ABB RobotStudio station: Modulo_2.rspag

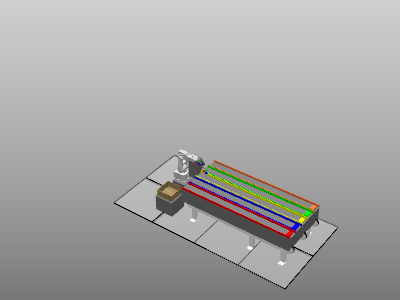
--- station ---
Station Project2 (saved by RobotStudio 25.1.11133.0)
Controller Controlador1, task T_ROB1: task frame (RAPID world) sits at (0, 0, 437.58) mm in the station
Controller Controlador1
  mechanical unit ROB_1: IRB120_3_58__01, 6 joints, base frame (0, 0, 0) mm
Layout (positions relative to the parent item):
  - IRB120_3_58__01 [mechanism, from %ABB.RobotStudio.Models.IRB120%\IRB120_3_58_G_01.rslib] at (0, 0, 437.58) mm; joint values [0, 0, 0, 0, 0.5236, 0] (rad or m)
  - MyTool [mechanism, from Training Objects\myTool.rslib] at (364.35, 0, 1031.58) mm, rotated rx 180 ry 60 rz 180 deg
  - Conveyor [part, from %ABB.RobotStudio.Models.Conveyors%\Conveyor 2400 3str h2.rslib] at (479.82, -405.8, 0) mm
  - Base Robot [graphiccomponentgroup]
    - Pieza_1 [part] at (-150, -150, 0) mm, size 300 x 300 x 200 mm
    - Pieza_2 [part], size 300 x 300 x 237.6 mm
  - Caja [part] at (0, 0, 145) mm, size 350 x 350 x 150 mm
  - Estropajo_Morado [part] at (2649.97, 391.91, 691.61) mm, size 80 x 120 x 43 mm
  - Estropajo_Verde [part] at (2649.97, 171.91, 691.61) mm, size 80 x 120 x 43 mm
  - Estropajo_Amarillo [part, from Components\Estropajo_6.rslib] at (2649.97, -48.09, 691.61) mm
  - Estropajo_Azul [part] at (2649.97, -268.09, 691.61) mm, size 80 x 120 x 43 mm
  - Estropajo_Rojo [part] at (2649.97, -488.09, 691.61) mm, size 80 x 120 x 43 mm
  - Base Caja [graphiccomponentgroup]
    - Base Caja [part] at (-190.34, -650.22, 0) mm, size 400 x 400 x 350 mm
  - LinearMover2 [smart component, from Components\LinearMover2.rslib]
      properties: Object=(none); Direction=[-0.001 0 0]; Distance=2.2; Duration=2; Reference=Global; ReferenceObject=(none)
  - LinearMover2_2 [smart component, from Components\LinearMover2.rslib]
      properties: Object=(none); Direction=[-0.001 0 0]; Distance=2.2; Duration=2; Reference=Global; ReferenceObject=(none)
  - LinearMover2_3 [smart component, from Components\LinearMover2.rslib]
      properties: Object=(none); Direction=[-0.001 0 0]; Distance=2.2; Duration=2; Reference=Global; ReferenceObject=(none)
  - LinearMover2_4 [smart component, from Components\LinearMover2.rslib]
      properties: Object=(none); Direction=[-0.001 0 0]; Distance=2.2; Duration=2; Reference=Global; ReferenceObject=(none)
  - LinearMover2_5 [smart component, from Components\LinearMover2.rslib]
      properties: Object=(none); Direction=[-0.001 0 0]; Distance=2.2; Duration=2; Reference=Global; ReferenceObject=(none)
  - Source [smart component, from Components\Source.rslib]
      properties: Source=Estropajo_Rojo; Copy=(none); Parent=(none); Position=[2.649968 -0.488094 0.691615]; Orientation=[0 0 0]; Transient=true; PhysicsBehavior=-1
  - Source_2 [smart component, from Components\Source.rslib]
      properties: Source=Estropajo_Azul; Copy=(none); Parent=(none); Position=[2.649968 -0.268094 0.691615]; Orientation=[0 0 0]; Transient=true; PhysicsBehavior=-1
  - Source_3 [smart component, from Components\Source.rslib]
      properties: Source=Estropajo_Amarillo; Copy=(none); Parent=(none); Position=[2.649968 -0.048094 0.691615]; Orientation=[0 0 0]; Transient=true; PhysicsBehavior=-1
  - Source_4 [smart component, from Components\Source.rslib]
      properties: Source=Estropajo_Verde; Copy=(none); Parent=(none); Position=[2.649968 0.171906 0.691615]; Orientation=[0 0 0]; Transient=true; PhysicsBehavior=-1
  - Source_5 [smart component, from Components\Source.rslib]
      properties: Source=Estropajo_Morado; Copy=(none); Parent=(none); Position=[2.649968 0.391906 0.691615]; Orientation=[0 0 0]; Transient=true; PhysicsBehavior=-1
  - Base Apilar [part], size 200 x 200 x 700 mm
  - Attacher [smart component, from Components\Attacher.rslib]
      properties: Parent=MyTool; Flange=0; Child=(none); Mount=false; Offset=[0 0 0]; Orientation=[0 0 0]
  - Attacher_2 [smart component, from Components\Attacher.rslib]
      properties: Parent=MyTool; Flange=0; Child=(none); Mount=false; Offset=[0 0 0]; Orientation=[0 0 0]
  - Attacher_3 [smart component, from Components\Attacher.rslib]
      properties: Parent=MyTool; Flange=0; Child=(none); Mount=false; Offset=[0 0 0]; Orientation=[0 0 0]
  - Attacher_4 [smart component, from Components\Attacher.rslib]
      properties: Parent=MyTool; Flange=0; Child=(none); Mount=false; Offset=[0 0 0]; Orientation=[0 0 0]
  - Attacher_5 [smart component, from Components\Attacher.rslib]
      properties: Parent=MyTool; Flange=0; Child=(none); Mount=false; Offset=[0 0 0]; Orientation=[0 0 0]
  - Detacher [smart component, from Components\Detacher.rslib]
      properties: Child=(none); KeepPosition=true
  - Detacher_2 [smart component, from Components\Detacher.rslib]
      properties: Child=(none); KeepPosition=true
  - Detacher_3 [smart component, from Components\Detacher.rslib]
      properties: Child=(none); KeepPosition=true
  - Detacher_4 [smart component, from Components\Detacher.rslib]
      properties: Child=(none); KeepPosition=true
  - Detacher_5 [smart component, from Components\Detacher.rslib]
      properties: Child=(none); KeepPosition=true
  - Cinta salida_2 [part, from Components\Cinta salida.rslib] at (2961.89, -775, 0) mm
Attachment: MyTool is attached to IRB120_3_58__01 / Link6
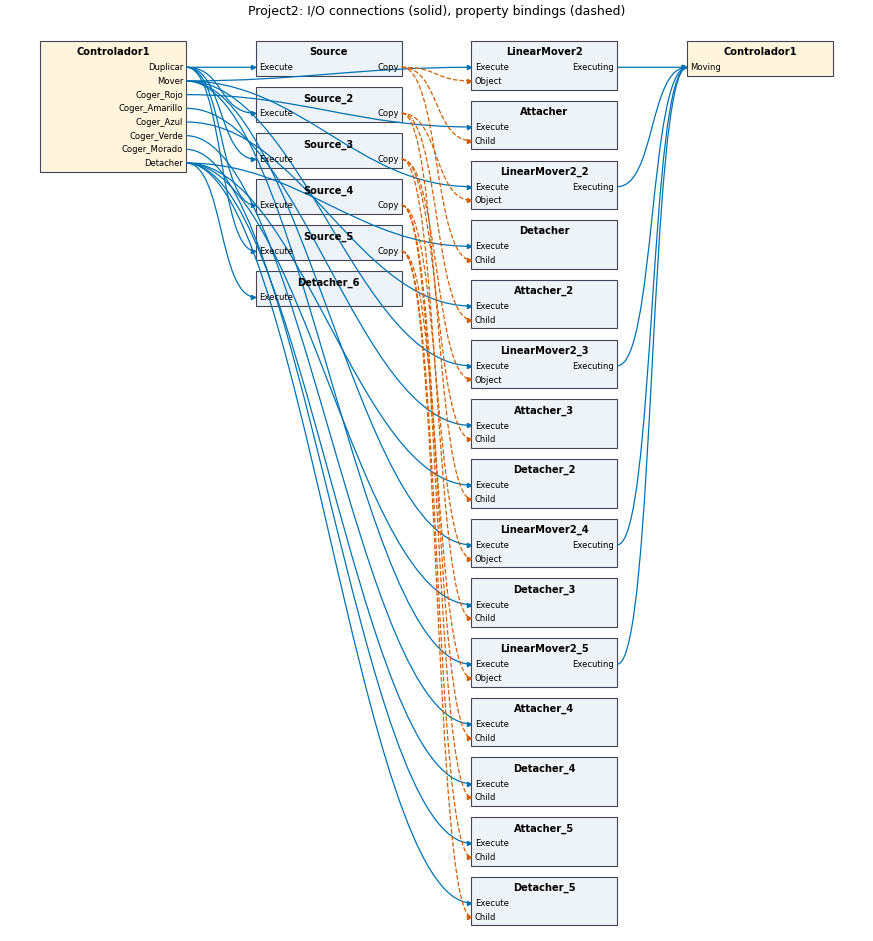
Station logic (signal -> signal, property => property):
  Controlador1.Duplicar -> Source.Execute
  Controlador1.Duplicar -> Source_2.Execute
  Controlador1.Duplicar -> Source_3.Execute
  Controlador1.Duplicar -> Source_4.Execute
  Controlador1.Duplicar -> Source_5.Execute
  Controlador1.Mover -> LinearMover2.Execute
  Controlador1.Mover -> LinearMover2_2.Execute
  Controlador1.Mover -> LinearMover2_3.Execute
  Controlador1.Mover -> LinearMover2_4.Execute
  Controlador1.Mover -> LinearMover2_5.Execute
  Controlador1.Coger_Rojo -> Attacher.Execute
  Controlador1.Coger_Amarillo -> Attacher_3.Execute
  Controlador1.Coger_Azul -> Attacher_2.Execute
  Controlador1.Coger_Verde -> Attacher_4.Execute
  Controlador1.Coger_Morado -> Attacher_5.Execute
  Controlador1.Detacher -> Detacher.Execute
  Controlador1.Detacher -> Detacher_2.Execute
  Controlador1.Detacher -> Detacher_3.Execute
  Controlador1.Detacher -> Detacher_4.Execute
  Controlador1.Detacher -> Detacher_5.Execute
  LinearMover2.Executing -> Controlador1.Moving
  LinearMover2_3.Executing -> Controlador1.Moving
  LinearMover2_5.Executing -> Controlador1.Moving
  LinearMover2_2.Executing -> Controlador1.Moving
  LinearMover2_4.Executing -> Controlador1.Moving
  Controlador1.Detacher -> Detacher_6.Execute
  Source.Copy => LinearMover2.Object
  Source_5.Copy => LinearMover2_5.Object
  Source_2.Copy => LinearMover2_2.Object
  Source_3.Copy => LinearMover2_3.Object
  Source_4.Copy => LinearMover2_4.Object
  Source_5.Copy => Attacher_5.Child
  Source_2.Copy => Attacher_2.Child
  Source_3.Copy => Attacher_3.Child
  Source_4.Copy => Attacher_4.Child
  Source.Copy => Attacher.Child
  Source_5.Copy => Detacher_5.Child
  Source_2.Copy => Detacher_2.Child
  Source.Copy => Detacher.Child
  Source_3.Copy => Detacher_3.Child
  Source_4.Copy => Detacher_4.Child

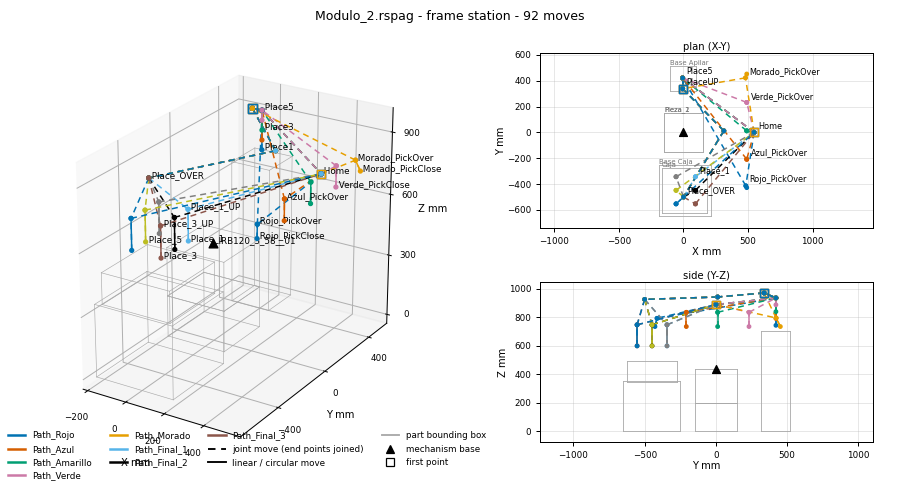
[picture p0: tool path of Modulo_2.rspag in frame station, 92 of 92 moves have a stored position in this frame; points joined in program order, loops and branches not executed]
--- Controller Data/Controlador1/RAPID/TASK1/PROGMOD/CalibData.mod ---
MODULE CalibData
    PERS tooldata MyTool:=[TRUE,[[31.7926,0,229.639],[0.945519,0,0.325568,0]],[1,[0,0,1],[1,0,0,0],0,0,0]];
ENDMODULE

--- Controller Data/Controlador1/RAPID/TASK1/PROGMOD/Module1.mod ---
MODULE Module1
    CONST robtarget Home:=[[547.330665099,0,451.64730631],[0.190808996,0,0.981627183,0],[0,0,0,0],[9E+09,9E+09,9E+09,9E+09,9E+09,9E+09]];
    CONST robtarget Rojo_PickOver:=[[482.707181756,-413.627425594,354.825525618],[0,0.382683432,0.923879533,0],[-1,-1,0,0],[9E+09,9E+09,9E+09,9E+09,9E+09,9E+09]];
    CONST robtarget Rojo_PickClose:=[[489.968,-428.094,297.038196778],[0,0.382683432,0.923879533,0],[0,0,0,0],[9E+09,9E+09,9E+09,9E+09,9E+09,9E+09]];
    CONST robtarget Place5:=[[-5.944,420.879,497.620196778],[0,0.923879533,-0.382683432,0],[1,-1,0,0],[9E+09,9E+09,9E+09,9E+09,9E+09,9E+09]];
    CONST robtarget Place1:=[[-5.944,420.879,305.620196778],[0,-0.382683432,0.923879533,0],[1,-1,0,0],[9E+09,9E+09,9E+09,9E+09,9E+09,9E+09]];
    CONST robtarget Azul_PickOver:=[[489.968,-208.094,397.038196778],[0,0.258819045,0.965925826,0],[-1,-1,0,0],[9E+09,9E+09,9E+09,9E+09,9E+09,9E+09]];
    CONST robtarget Azul_PickClose:=[[489.968,-208.094,297.038196778],[0,0.258819045,0.965925826,0],[-1,-1,0,0],[9E+09,9E+09,9E+09,9E+09,9E+09,9E+09]];
    CONST robtarget Place2:=[[-5.944,420.879,353.620196778],[0,-0.5,0.866025404,0],[1,-1,0,0],[9E+09,9E+09,9E+09,9E+09,9E+09,9E+09]];
    CONST robtarget Amarillo_PickOver:=[[489.968,11.906,397.038196778],[0,0,1,0],[0,-1,0,0],[9E+09,9E+09,9E+09,9E+09,9E+09,9E+09]];
    CONST robtarget Amarillo_PickClose:=[[489.968,11.906,297.038196778],[0,0,1,0],[0,-1,0,0],[9E+09,9E+09,9E+09,9E+09,9E+09,9E+09]];
    CONST robtarget Place3:=[[-5.944,420.879,401.620196778],[0,-0.707106781,0.707106781,0],[1,-1,0,0],[9E+09,9E+09,9E+09,9E+09,9E+09,9E+09]];
    CONST robtarget Verde_PickOver:=[[489.968,231.906,397.038196778],[0,-0.258819045,0.965925826,0],[0,0,-1,0],[9E+09,9E+09,9E+09,9E+09,9E+09,9E+09]];
    CONST robtarget Verde_PickClose:=[[489.968,231.906,297.038196778],[0,-0.258819045,0.965925826,0],[0,0,-1,0],[9E+09,9E+09,9E+09,9E+09,9E+09,9E+09]];
    CONST robtarget Place4:=[[-5.944,420.879,449.620196778],[0,0.866025404,-0.5,0],[1,-1,0,0],[9E+09,9E+09,9E+09,9E+09,9E+09,9E+09]];
    CONST robtarget Morado_PickOver:=[[480.242120381,422.191842909,357.360002191],[0,-0.382683432,0.923879533,0],[0,0,0,0],[9E+09,9E+09,9E+09,9E+09,9E+09,9E+09]];
    CONST robtarget Morado_PickClose:=[[489.968,451.906,297.038196778],[0,-0.382683432,0.923879533,0],[0,0,-1,0],[9E+09,9E+09,9E+09,9E+09,9E+09,9E+09]];
    CONST robtarget PlaceUP:=[[-5.944,337.901122968,532.92991778],[0,0.923879532,-0.382683433,0],[1,-1,0,0],[9E+09,9E+09,9E+09,9E+09,9E+09,9E+09]];
    CONST robtarget PlaceUP_2:=[[-5.944,337.901122968,532.92991778],[0,-0.707106781,0.707106782,0],[1,-1,0,0],[9E+09,9E+09,9E+09,9E+09,9E+09,9E+09]];
    CONST robtarget Place5_2:=[[-5.944,420.879,497.620196778],[0,0.707106782,-0.707106781,0],[1,-1,0,0],[9E+09,9E+09,9E+09,9E+09,9E+09,9E+09]];
    CONST robtarget Place_1_UP:=[[92.759,-343.568,309.203196778],[0,0.707106781,0.707106781,0],[-1,-1,0,0],[9E+09,9E+09,9E+09,9E+09,9E+09,9E+09]];
    CONST robtarget Place_1:=[[92.759,-343.568,161.203196778],[0,0.707106781,0.707106781,0],[-1,-1,0,0],[9E+09,9E+09,9E+09,9E+09,9E+09,9E+09]];
    CONST robtarget Place_2_UP:=[[92.759,-448.568,309.203196778],[0,0.707106781,0.707106781,0],[-1,-1,0,0],[9E+09,9E+09,9E+09,9E+09,9E+09,9E+09]];
    CONST robtarget Place_2:=[[92.759,-448.568,161.203196778],[0,0.707106781,0.707106781,0],[-1,-1,0,0],[9E+09,9E+09,9E+09,9E+09,9E+09,9E+09]];
    CONST robtarget Place_3_UP:=[[92.759,-553.568,309.203196778],[0,0.707106781,0.707106781,0],[-1,-1,0,0],[9E+09,9E+09,9E+09,9E+09,9E+09,9E+09]];
    CONST robtarget Place_3:=[[92.759,-553.568,161.203196778],[0,0.707106781,0.707106781,0],[-1,-1,0,0],[9E+09,9E+09,9E+09,9E+09,9E+09,9E+09]];
    CONST robtarget Place_4_UP:=[[-57.241,-343.568,309.203196778],[0,0.707106781,0.707106781,0],[-2,0,-1,0],[9E+09,9E+09,9E+09,9E+09,9E+09,9E+09]];
    CONST robtarget Place_4:=[[-57.241,-343.568,161.203196778],[0,0.707106781,0.707106781,0],[-2,0,-1,0],[9E+09,9E+09,9E+09,9E+09,9E+09,9E+09]];
    CONST robtarget Place_5_UP:=[[-57.241,-448.568,309.203196778],[0,0.707106781,0.707106781,0],[-2,0,-1,0],[9E+09,9E+09,9E+09,9E+09,9E+09,9E+09]];
    CONST robtarget Place_5:=[[-57.241,-448.568,161.203196778],[0,0.707106781,0.707106781,0],[-2,0,-1,0],[9E+09,9E+09,9E+09,9E+09,9E+09,9E+09]];
    CONST robtarget Place_6_UP:=[[-57.241,-553.568,309.203196778],[0,0.707106781,0.707106781,0],[-2,0,-1,0],[9E+09,9E+09,9E+09,9E+09,9E+09,9E+09]];
    CONST robtarget Place_6:=[[-57.241,-553.568,161.203196778],[0,0.707106781,0.707106781,0],[-2,0,-1,0],[9E+09,9E+09,9E+09,9E+09,9E+09,9E+09]];
    CONST robtarget Place_MEDIO:=[[312.75,11.906,504.639984673],[0,0,1,0],[0,-1,0,0],[9E+09,9E+09,9E+09,9E+09,9E+09,9E+09]];
    CONST robtarget Place_OVER:=[[0.756047431,-500.595624659,487.67995873],[0,0.707106781,0.707106781,0],[-1,-1,0,0],[9E+09,9E+09,9E+09,9E+09,9E+09,9E+09]];

    PROC main()
        PulseDO Duplicar;
        PulseDO Mover;
        WaitUntil Moving = 1;
        WaitUntil Moving = 0;

        Path_Apilar;
        Path_Final_1;

        PulseDO Duplicar;
        PulseDO Mover;
        WaitUntil Moving = 1;
        WaitUntil Moving = 0;

        Path_Apilar;
        Path_Final_2;

        PulseDO Duplicar;
        PulseDO Mover;
        WaitUntil Moving = 1;
        WaitUntil Moving = 0;

        Path_Apilar;
        Path_Final_3;

        PulseDO Duplicar;
        PulseDO Mover;
        WaitUntil Moving = 1;
        WaitUntil Moving = 0;

        Path_Apilar;
        Path_Final_4;

        PulseDO Duplicar;
        PulseDO Mover;
        WaitUntil Moving = 1;
        WaitUntil Moving = 0;

        Path_Apilar;
        Path_Final_5;

        PulseDO Duplicar;
        PulseDO Mover;
        WaitUntil Moving = 1;
        WaitUntil Moving = 0;

        Path_Apilar;
        Path_Final_6;
    ENDPROC

    PROC Path_Apilar()
        SetDO Coger_Rojo, 0;
        SetDO Coger_Azul, 0;
        SetDO Coger_Amarillo, 0;
        SetDO Coger_Verde, 0;
        SetDO Coger_Morado, 0;
        PulseDO Detacher;
        Path_Rojo;
        Path_Azul;
        Path_Amarillo;
        Path_Verde;
        Path_Morado;
    ENDPROC

    PROC Path_Rojo()
        MoveJ Home,v1000,fine,MyTool\WObj:=wobj0;
        MoveJ Rojo_PickOver,v1000,fine,MyTool\WObj:=wobj0;
        MoveL Rojo_PickClose,v300,fine,MyTool\WObj:=wobj0;
        SetDO Coger_Rojo, 1;
        MoveJ Rojo_PickOver,v1000,fine,MyTool\WObj:=wobj0;
        MoveJ Place5,v1000,fine,MyTool\WObj:=wobj0;
        MoveL Place1,v300,fine,MyTool\WObj:=wobj0;
        SetDO Coger_Rojo, 0;
        PulseDO Detacher;
        MoveJ Place5,v1000,fine,MyTool\WObj:=wobj0;
        MoveJ Home,v1000,fine,MyTool\WObj:=wobj0;
    ENDPROC

    PROC Path_Azul()
        MoveJ Home,v1000,fine,MyTool\WObj:=wobj0;
        MoveJ Azul_PickOver,v1000,fine,MyTool\WObj:=wobj0;
        MoveL Azul_PickClose,v300,fine,MyTool\WObj:=wobj0;
        SetDO Coger_Azul, 1;
        MoveJ Azul_PickOver,v1000,fine,MyTool\WObj:=wobj0;
        MoveJ Place5,v1000,fine,MyTool\WObj:=wobj0;
        MoveL Place2,v300,fine,MyTool\WObj:=wobj0;
        SetDO Coger_Azul, 0;
        PulseDO Detacher;
        MoveJ Place5,v1000,fine,MyTool\WObj:=wobj0;
        MoveJ Home,v1000,fine,MyTool\WObj:=wobj0;
    ENDPROC

    PROC Path_Amarillo()
        MoveJ Home,v1000,z0,MyTool\WObj:=wobj0;
        MoveJ Amarillo_PickOver,v1000,z0,MyTool\WObj:=wobj0;
        MoveL Amarillo_PickClose,v300,z0,MyTool\WObj:=wobj0;
        WaitTime 0.5;
        SetDO Coger_Amarillo, 1;
        MoveJ Amarillo_PickOver,v1000,z0,MyTool\WObj:=wobj0;
        MoveJ Place5,v1000,z0,MyTool\WObj:=wobj0;
        MoveL Place3,v300,z0,MyTool\WObj:=wobj0;
        WaitTime 0.7;
        SetDO Coger_Amarillo, 0;
        PulseDO Detacher;
        MoveJ Place5,v1000,fine,MyTool\WObj:=wobj0;
        MoveJ Home,v1000,z0,MyTool\WObj:=wobj0;
    ENDPROC

    PROC Path_Verde()
        MoveJ Home,v1000,fine,MyTool\WObj:=wobj0;
        MoveJ Verde_PickOver,v1000,fine,MyTool\WObj:=wobj0;
        MoveL Verde_PickClose,v200,fine,MyTool\WObj:=wobj0;
        SetDO Coger_Verde, 1;
        MoveJ Verde_PickOver,v1000,fine,MyTool\WObj:=wobj0;
        MoveJ Place5,v1000,fine,MyTool\WObj:=wobj0;
        MoveL Place4,v200,fine,MyTool\WObj:=wobj0;
        SetDO Coger_Verde, 0;
        PulseDO Detacher;
        MoveJ Place5,v1000,fine,MyTool\WObj:=wobj0;
        MoveJ Home,v1000,fine,MyTool\WObj:=wobj0;
    ENDPROC

    PROC Path_Morado()
        MoveJ Home,v1000,z0,MyTool\WObj:=wobj0;
        MoveJ Morado_PickOver,v1000,z0,MyTool\WObj:=wobj0;
        MoveL Morado_PickClose,v300,fine,MyTool\WObj:=wobj0;
        SetDO Coger_Morado, 1;
        MoveJ Morado_PickOver,v1000,z0,MyTool\WObj:=wobj0;
        MoveJ PlaceUP,v1000,z0,MyTool\WObj:=wobj0;
        MoveL Place5,v300,fine,MyTool\WObj:=wobj0;
        SetDO Coger_Morado, 0;
        PulseDO Detacher;
    ENDPROC

    PROC Path_Final_1()
        MoveJ PlaceUP_2,v1000,fine,MyTool\WObj:=wobj0;
        MoveL Place5_2,v200,fine,MyTool\WObj:=wobj0;
        WaitTime 0.5;
        SetDO Coger_Rojo, 1;
        SetDO Coger_Azul, 1;
        SetDO Coger_Amarillo, 1;
        SetDO Coger_Verde, 1;
        SetDO Coger_Morado, 1;
        MoveJ PlaceUP_2,v1000,fine,MyTool\WObj:=wobj0;
        MoveJ Place_MEDIO,v1000,fine,MyTool\WObj:=wobj0;
        MoveJ Place_OVER,v1000,fine,MyTool\WObj:=wobj0;
        MoveJ Place_1_UP,v1000,fine,MyTool\WObj:=wobj0;
        MoveL Place_1,v150,fine,MyTool\WObj:=wobj0;
        WaitTime 0.5;
        SetDO Coger_Rojo, 0;
        SetDO Coger_Azul, 0;
        SetDO Coger_Amarillo, 0;
        SetDO Coger_Verde, 0;
        SetDO Coger_Morado, 0;
        PulseDO Detacher;
        MoveJ Place_1_UP,v1000,fine,MyTool\WObj:=wobj0;
        MoveJ Home,v1000,fine,MyTool\WObj:=wobj0;
    ENDPROC

    PROC Path_Final_2()
        MoveJ PlaceUP_2,v1000,fine,MyTool\WObj:=wobj0;
        MoveL Place5_2,v200,fine,MyTool\WObj:=wobj0;
        WaitTime 0.5;
        SetDO Coger_Rojo, 1;
        SetDO Coger_Azul, 1;
        SetDO Coger_Amarillo, 1;
        SetDO Coger_Verde, 1;
        SetDO Coger_Morado, 1;
        MoveJ PlaceUP_2,v1000,fine,MyTool\WObj:=wobj0;
        MoveJ Place_MEDIO,v1000,fine,MyTool\WObj:=wobj0;
        MoveJ Place_OVER,v1000,fine,MyTool\WObj:=wobj0;
        MoveJ Place_2_UP,v1000,fine,MyTool\WObj:=wobj0;
        MoveL Place_2,v200,fine,MyTool\WObj:=wobj0;
        WaitTime 0.5;
        SetDO Coger_Rojo, 0;
        SetDO Coger_Azul, 0;
        SetDO Coger_Amarillo, 0;
        SetDO Coger_Verde, 0;
        SetDO Coger_Morado, 0;
        PulseDO Detacher;
        MoveJ Place_2_UP,v1000,fine,MyTool\WObj:=wobj0;
        MoveJ Home,v1000,fine,MyTool\WObj:=wobj0;
    ENDPROC

    PROC Path_Final_3()
        MoveJ PlaceUP_2,v1000,fine,MyTool\WObj:=wobj0;
        MoveL Place5_2,v200,fine,MyTool\WObj:=wobj0;
        WaitTime 0.5;
        SetDO Coger_Rojo, 1;
        SetDO Coger_Azul, 1;
        SetDO Coger_Amarillo, 1;
        SetDO Coger_Verde, 1;
        SetDO Coger_Morado, 1;
        MoveJ PlaceUP_2,v1000,fine,MyTool\WObj:=wobj0;
        MoveJ Place_MEDIO,v1000,fine,MyTool\WObj:=wobj0;
        MoveJ Place_OVER,v1000,fine,MyTool\WObj:=wobj0;
        MoveJ Place_3_UP,v1000,fine,MyTool\WObj:=wobj0;
        MoveL Place_3,v200,fine,MyTool\WObj:=wobj0;
        WaitTime 0.5;
        SetDO Coger_Rojo, 0;
        SetDO Coger_Azul, 0;
        SetDO Coger_Amarillo, 0;
        SetDO Coger_Verde, 0;
        SetDO Coger_Morado, 0;
        PulseDO Detacher;
        MoveJ Place_3_UP,v1000,fine,MyTool\WObj:=wobj0;
        MoveJ Home,v1000,fine,MyTool\WObj:=wobj0;
    ENDPROC

    PROC Path_Final_4()
        MoveJ PlaceUP_2,v1000,fine,MyTool\WObj:=wobj0;
        MoveL Place5_2,v200,fine,MyTool\WObj:=wobj0;
        WaitTime 0.5;
        SetDO Coger_Rojo, 1;
        SetDO Coger_Azul, 1;
        SetDO Coger_Amarillo, 1;
        SetDO Coger_Verde, 1;
        SetDO Coger_Morado, 1;
        MoveJ PlaceUP_2,v1000,fine,MyTool\WObj:=wobj0;
        MoveJ Place_MEDIO,v1000,fine,MyTool\WObj:=wobj0;
        MoveJ Place_OVER,v1000,fine,MyTool\WObj:=wobj0;
        MoveJ Place_4_UP,v1000,fine,MyTool\WObj:=wobj0;
        MoveL Place_4,v200,fine,MyTool\WObj:=wobj0;
        WaitTime 0.5;
        SetDO Coger_Rojo, 0;
        SetDO Coger_Azul, 0;
        SetDO Coger_Amarillo, 0;
        SetDO Coger_Verde, 0;
        SetDO Coger_Morado, 0;
        PulseDO Detacher;
        MoveJ Place_4_UP,v1000,fine,MyTool\WObj:=wobj0;
        MoveJ Home,v1000,fine,MyTool\WObj:=wobj0;
    ENDPROC

    PROC Path_Final_5()
        MoveJ PlaceUP_2,v1000,fine,MyTool\WObj:=wobj0;
        MoveL Place5_2,v200,fine,MyTool\WObj:=wobj0;
        WaitTime 0.5;
        SetDO Coger_Rojo, 1;
        SetDO Coger_Azul, 1;
        SetDO Coger_Amarillo, 1;
        SetDO Coger_Verde, 1;
        SetDO Coger_Morado, 1;
        MoveJ PlaceUP_2,v1000,fine,MyTool\WObj:=wobj0;
        MoveJ Place_MEDIO,v1000,fine,MyTool\WObj:=wobj0;
        MoveJ Place_OVER,v1000,fine,MyTool\WObj:=wobj0;
        MoveJ Place_5_UP,v1000,fine,MyTool\WObj:=wobj0;
        MoveL Place_5,v200,fine,MyTool\WObj:=wobj0;
        WaitTime 0.5;
        SetDO Coger_Rojo, 0;
        SetDO Coger_Azul, 0;
        SetDO Coger_Amarillo, 0;
        SetDO Coger_Verde, 0;
        SetDO Coger_Morado, 0;
        PulseDO Detacher;
        MoveJ Place_5_UP,v1000,fine,MyTool\WObj:=wobj0;
        MoveJ Home,v1000,fine,MyTool\WObj:=wobj0;
    ENDPROC

    PROC Path_Final_6()
        MoveJ PlaceUP_2,v1000,fine,MyTool\WObj:=wobj0;
        MoveL Place5_2,v200,fine,MyTool\WObj:=wobj0;
        WaitTime 0.5;
        SetDO Coger_Rojo, 1;
        SetDO Coger_Azul, 1;
        SetDO Coger_Amarillo, 1;
        SetDO Coger_Verde, 1;
        SetDO Coger_Morado, 1;
        MoveJ PlaceUP_2,v1000,fine,MyTool\WObj:=wobj0;
        MoveJ Place_MEDIO,v1000,fine,MyTool\WObj:=wobj0;
        MoveJ Place_OVER,v1000,fine,MyTool\WObj:=wobj0;
        MoveJ Place_6_UP,v1000,fine,MyTool\WObj:=wobj0;
        MoveL Place_6,v200,fine,MyTool\WObj:=wobj0;
        WaitTime 0.5;
        SetDO Coger_Rojo, 0;
        SetDO Coger_Azul, 0;
        SetDO Coger_Amarillo, 0;
        SetDO Coger_Verde, 0;
        SetDO Coger_Morado, 0;
        PulseDO Detacher;
        MoveJ Place_6_UP,v1000,fine,MyTool\WObj:=wobj0;
        MoveJ Home,v1000,fine,MyTool\WObj:=wobj0;
    ENDPROC

ENDMODULE

--- Controller Data/Controlador1/SYSPAR/EIO.cfg ---
EIO:CFG_1.0:6:1::
#
EIO_SIGNAL:

      -Name "Duplicar" -SignalType "DO" -Access "All"

      -Name "Mover" -SignalType "DO" -Access "All"

      -Name "Coger_Rojo" -SignalType "DO" -Access "All"

      -Name "Coger_Amarillo" -SignalType "DO" -Access "All"

      -Name "Coger_Azul" -SignalType "DO" -Access "All"

      -Name "Coger_Verde" -SignalType "DO" -Access "All"

      -Name "Coger_Morado" -SignalType "DO" -Access "All"

      -Name "Detacher" -SignalType "DO" -Access "All"

      -Name "Moving" -SignalType "DI" -Access "All"
